PROGRAM MAIN
VAR
	Comm	: FB_Comm_MQTT_Influx;
END_VAR

Comm(
	sHostName	:= '',
	nHostPort	:= 0,
	nKeepAlive	:= 0,
	sTopicSub	:= '');

END_PROGRAM

(* stored: Version 1.1.0.1, ProductVersion 3.1.4024.13
   POU MAIN: Id {6cfeea34-4fca-49d7-9b7c-57f77e87b2d0}, SpecialFunc None *)
